{attribute addProperty BoxType "EK1100-0000-0018"}
{attribute addProperty Id "Beckhoff_EJ4xxxEK1122Beckhoff_EJ4xxxEK1122_15AA3F2B162A_0001_EJ4002_0000_0017EJ4002_08E1E1D812015A_0002_EJ4002_0000_0018EJ4002_F05A29F112015A_0003_EJ4004_0000_0020EJ4004_253CF8AE15219A_0004_EJ4008_0000_0020EJ4008_E04CC7BF21627A_0005_EJ4018_0000_0016EJ4018_E04CC7BF21627A_0006_EJ4024_0000_0020EJ4024_253CF8AE15219A_0007_EJ4132_0000_0019EJ4132_08E1E1D812015A_0008_EJ4134_0000_0019EJ4134_57EE2D9D15219A_0009_EJ4134_0000_0020EJ4134_57EE2D9D15219"}
{attribute addProperty CRC "2483289938"}
{attribute addProperty SizeInBites "1416"}
{attribute addProperty SizeInBytes "177"}
TYPE Beckhoff_EJ4xxx_9403FF52 EXTENDS EK1100_179A0949 :
STRUCT
	{attribute addProperty Name "Beckhoff_EJ4xxxEK1122"}
	Beckhoff_EJ4xxxEK1122 : Beckhoff_EJ4xxxEK1122_15AA3F2B;
	{attribute addProperty Name "A_0001_EJ4002_0000_0017"}
	A_0001_EJ4002_0000_0017 : EJ4002_08E1E1D8;
	{attribute addProperty Name "A_0002_EJ4002_0000_0018"}
	A_0002_EJ4002_0000_0018 : EJ4002_F05A29F1;
	{attribute addProperty Name "A_0003_EJ4004_0000_0020"}
	A_0003_EJ4004_0000_0020 : EJ4004_253CF8AE;
	{attribute addProperty Name "A_0004_EJ4008_0000_0020"}
	A_0004_EJ4008_0000_0020 : EJ4008_E04CC7BF;
	{attribute addProperty Name "A_0005_EJ4018_0000_0016"}
	A_0005_EJ4018_0000_0016 : EJ4018_E04CC7BF;
	{attribute addProperty Name "A_0006_EJ4024_0000_0020"}
	A_0006_EJ4024_0000_0020 : EJ4024_253CF8AE;
	{attribute addProperty Name "A_0007_EJ4132_0000_0019"}
	A_0007_EJ4132_0000_0019 : EJ4132_08E1E1D8;
	{attribute addProperty Name "A_0008_EJ4134_0000_0019"}
	A_0008_EJ4134_0000_0019 : EJ4134_57EE2D9D;
	{attribute addProperty Name "A_0009_EJ4134_0000_0020"}
	A_0009_EJ4134_0000_0020 : EJ4134_57EE2D9D;
END_STRUCT
END_TYPE

(* stored: Version 1.2.0.0, ProductVersion 3.1.4024.9
   DUT Beckhoff_EJ4xxx_9403FF52: Id {28384b39-e540-46b0-804c-79c49d7630e4} *)
